# EPICS alarm handler configuration: mps_database/bareTest/alarms/areas/mpln_ltuh_mp05.alhConfig
GROUP NULL MPLN:LTUH:MP05:1
$ALIAS MPS Link Node 134
$GUIDANCE
LTUH MPS
   Group Name: MPLN:LTUH:MP05:1
   Summary PV:  MPLN:LTUH:MP05:1:STATSUMY
$END
CHANNEL  MPLN:LTUH:MP05:1    MPLN:LTUH:MP05:1:MPS_EN_RBV		-----
CHANNEL  MPLN:LTUH:MP05:1    MPLN:LTUH:MP05:1:LC1_MODE_RBV		-----
